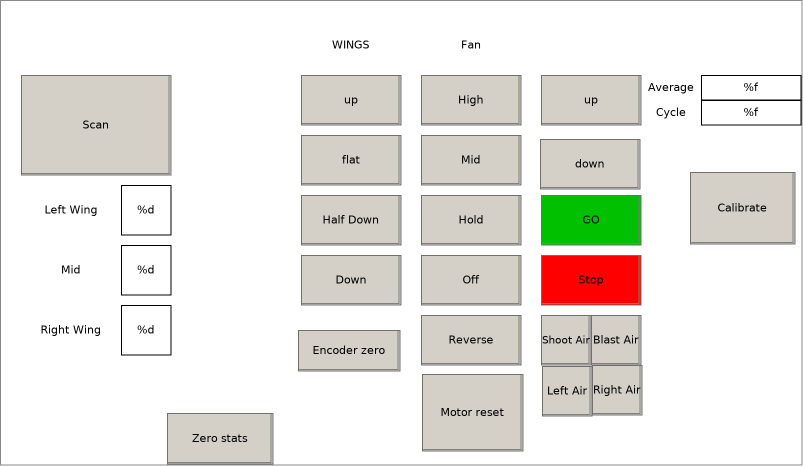
VISUALIZATION Visualization  // 803x466
    Button (422,374 101x77), "Motor reset"
        OnMouseDown: execute { GVL.ResetMotor :=TRUE; }
        OnMouseUp: execute { GVL.ResetMotor :=FALSE; }
    Button (21,75 150x100), "Scan"
        OnMouseDown: execute { GVL.ArduinoState := MAIN.Scanner; }
    Button (301,75 100x50), "up"
        OnMouseDown: execute { GVL.FanDyno :=MAIN.WingUp GVL.ArduinoState := MAIN.WingGo }
    Button (301,135 100x50), "flat"
        OnMouseDown: execute { GVL.FanDyno := MAIN.WingFlat GVL.ArduinoState := MAIN.WingGo }
    Button (301,255 100x50), "Down"
        OnMouseDown: execute { GVL.FanDyno :=MAIN.WingDown GVL.ArduinoState := MAIN.WingGo }
    Button (301,195 100x50), "Half Down"
        OnMouseDown: execute { GVL.FanDyno :=MAIN.WingHDown GVL.ArduinoState := MAIN.WingGo }
    Label (301,20 100x50), "WINGS"
    Button (421,75 100x50), "High"
        OnMouseDown: execute { GVL.FanDyno :=103 GVL.ArduinoState := MAIN.FanGo }
    Button (421,135 100x50), "Mid"
        OnMouseDown: execute { GVL.FanDyno :=100 GVL.ArduinoState := MAIN.FanGo }
    Button (421,255 100x50), "Off"
        OnMouseDown: execute { GVL.FanDyno :=89 GVL.ArduinoState := MAIN.FanGo }
    Button (421,195 100x50), "Hold"
        OnMouseDown: execute { GVL.FanDyno :=97 GVL.ArduinoState := MAIN.FanGo }
    Label (421,20 100x50), "Fan"
    Button (421,315 100x50), "Reverse"
        OnMouseDown: execute { GVL.FanDyno :=74 GVL.ArduinoState := MAIN.FanGo }
    Button (541,195 100x50), "GO"
        OnMouseUp: execute { MAIN.State := 100; MAIN.GoTime := MAIN.TimeSeconds; }
    Button (541,255 100x50), "Stop"
        OnMouseDown: execute {
            MAIN.State := 0;
            GVL.ArduinoState := 0;
            GVL.StepperUp := FALSE;
            GVL.StepperDown := FALSE;
            GVL.AirJet1 := FALSE;
            GVL.AirJet2 := FALSE;
            GVL.LeftAirJet := FALSE;
            GVL.RightAirJet := FALSE;
            GVL.VelocityMotor :=0;
            MAIN.TotalTime := MAIN.TimeSeconds;
        }
    Button (541,315 50x50), "Shoot Air"
        OnMouseDown: execute { GVL.AirJet2 := TRUE; }
        OnMouseUp: execute { GVL.AirJet2 := FALSE; }
    Button (591,315 50x50), "Blast Air"
        OnMouseDown: execute { GVL.AirJet1 := TRUE; }
        OnMouseUp: execute { GVL.AirJet1 := FALSE; }
    Button (541,75 100x50), "up"
        OnMouseDown: execute { GVL.StepperUp	:= TRUE; }
        OnMouseUp: execute { GVL.StepperUp	:= FALSE; GVL.VelocityMotor :=0; }
    Button (540,139 100x50), "down"
        OnMouseDown: execute { GVL.StepperDown	:= TRUE; }
        OnMouseUp: execute { GVL.StepperDown	:= FALSE; GVL.VelocityMotor :=0; }
    Rectangle (701,75 100x25), "%f", text variable: MAIN.AverageTime
    Rectangle (701,100 100x25), "%f", text variable: MAIN.CycleTime
    Label (621,75 100x25), "Average"
    Label (621,100 100x25), "Cycle"
    Button (690,172 105x72), "Calibrate"
        OnMouseDown: execute {
            MAIN.Calibrate := TRUE;
            MAIN.State := 100;
            MAIN.GoTime := MAIN.TimeSeconds;
        }
    Rectangle (121,185 50x50), "%d", text variable: MAIN.AverageLeft
    Rectangle (121,245 50x50), "%d", text variable: MAIN.Average
    Rectangle (121,305 50x50), "%d", text variable: MAIN.AverageRight
    Label (21,185 100x50), "Left Wing"
    Label (21,245 100x50), "Mid"
    Label (21,305 100x50), "Right Wing"
    Button (298,330 102x41), "Encoder zero"
        OnMouseDown: execute { GVL.SetCounterVal :=5000000; GVL.SetCounter :=TRUE; }
        OnMouseUp: execute {
            //ShooterBob.EncoderCount :=FALSE;
        }
    Button (542,366 50x50), "Left Air"
        OnMouseDown: execute { GVL.LeftAirJet := TRUE; }
        OnMouseUp: execute { GVL.LeftAirJet := FALSE; }
    Button (592,365 50x50), "Right Air"
        OnMouseDown: execute { GVL.RightAirJet := TRUE; }
        OnMouseUp: execute { GVL.RightAirJet := FALSE; }
    Button (167,413 106x51), "Zero stats"
        OnMouseDown: execute {
            MAIN.Singles :=0;
            MAIN.Doubles :=0;
            MAIN.Wiggle :=0;
            MAIN.Zeros :=0;
            MAIN.AverageTime :=0;
            MAIN.CycleTime := 0;
            MAIN.GoTime := 0;
            MAIN.EndTime  := 0;
            MAIN.StartTime := 0;
        }
END_VISUALIZATION

(* stored: Version 1.1.0.1, ProductVersion 3.1.4024.0
   Visu Visualization: Id {c6a0c5e7-ccfd-460e-88df-0ee3601afd8d} *)
